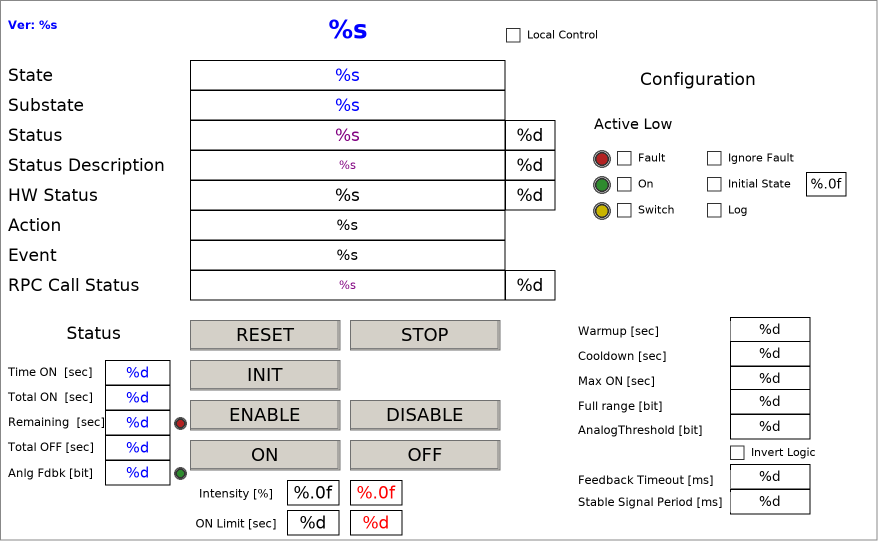
VISUALIZATION GUI_TEMPLATE_LAMP  // 878x541
VAR_IN_OUT
	m_Instance:	FB_LAMP;
END_VAR
    Rectangle (190,60 315x30), "%s", text variable: m_Instance.stat.sState
    Rectangle (190,90 315x30), "%s", text variable: m_Instance.stat.sSubstate
    Button (190,320 150x30), "RESET", input disabled if: (m_Instance.stat.bLocal = FALSE) <> 0
        OnMouseDown: execute { m_Instance.ctrl.nCommand := E_LAMP_COMMAND.RESET; m_Instance.ctrl.bExecute := TRUE; }
    Button (190,360 150x30), "INIT", input disabled if: (m_Instance.stat.bLocal = FALSE) <> 0
        OnMouseDown: execute { m_Instance.ctrl.nCommand := E_LAMP_COMMAND.INIT; m_Instance.ctrl.bExecute := TRUE; }
    Button (350,320 150x30), "STOP", input disabled if: (m_Instance.stat.bLocal = FALSE) <> 0
        OnMouseDown: execute { m_Instance.ctrl.nCommand := E_LAMP_COMMAND.STOP; m_Instance.ctrl.bExecute := TRUE; }
    Button (190,400 150x30), "ENABLE", input disabled if: (m_Instance.stat.bLocal = FALSE) <> 0
        OnMouseDown: execute { m_Instance.ctrl.nCommand := E_LAMP_COMMAND.ENABLE; m_Instance.ctrl.bExecute := TRUE; }
    Button (350,400 150x30), "DISABLE", input disabled if: (m_Instance.stat.bLocal = FALSE) <> 0
        OnMouseDown: execute { m_Instance.ctrl.nCommand := E_LAMP_COMMAND.DISABLE; m_Instance.ctrl.bExecute := TRUE; }
    Button (190,440 150x30), "ON", input disabled if: (m_Instance.stat.bLocal = FALSE) <> 0
        OnMouseDown: execute { m_Instance.ctrl.nCommand := E_LAMP_COMMAND.ON; m_Instance.ctrl.bExecute := TRUE; }
    Button (350,440 150x30), "OFF", input disabled if: (m_Instance.stat.bLocal = FALSE) <> 0
        OnMouseDown: execute { m_Instance.ctrl.nCommand := E_LAMP_COMMAND.OFF; m_Instance.ctrl.bExecute := TRUE; }
    Rectangle (5,60 180x30), "State"
    Rectangle (5,90 180x30), "Substate"
    Rectangle (190,120 315x30), "%s", text variable: m_Instance.stat.sStatus
    Rectangle (190,150 315x30), "%s", text variable: m_Instance.stat.sErrorText
    Rectangle (5,120 180x30), "Status"
    Rectangle (5,150 180x30), "Status Description"
    Rectangle (190,210 315x30), "%s", text variable: m_Instance.stat.sActionDesc
    Rectangle (190,240 315x30), "%s", text variable: m_Instance.stat.sEventDesc
    Rectangle (190,180 315x30), "%s", text variable: m_Instance.stat.sHwStatus
    Rectangle (5,180 180x30), "HW Status"
    Rectangle (505,180 50x30), "%d", text variable: m_Instance.stat.nHwStatus
    Rectangle (5,210 180x30), "Action"
    Rectangle (5,240 180x30), "Event"
    Rectangle (232,12 232x35), "%s", text variable: m_Instance.cfg.sName
    Rectangle (637,64 180x30), "Configuration"
    Rectangle (591,109 126x30), "Active Low"
    Checkbox (615,143 72x30), "Fault", variable: m_Instance.cfg.bActiveLowFault, input disabled if: (m_Instance.stat.bLocal = FALSE) <> 0
    Checkbox (705,143 102x30), "Ignore Fault", variable: m_Instance.cfg.bIgnoreFault, input disabled if: (m_Instance.stat.bLocal = FALSE) <> 0
    Checkbox (615,169 72x30), "On", variable: m_Instance.cfg.bActiveLowOn, input disabled if: (m_Instance.stat.bLocal = FALSE) <> 0
    Checkbox (615,195 72x30), "Switch", variable: m_Instance.cfg.bActiveLowSwitch, input disabled if: (m_Instance.stat.bLocal = FALSE) <> 0
    Checkbox (728,440 150x25), "Invert Logic", tooltip "If the logic is inverted, the lamp is considered to be ON, if the reading is below the threshold.", variable: m_Instance.cfg.bInvertAnalog, input disabled if: (m_Instance.stat.bLocal = FALSE) <> 0
    Rectangle (730,317 80x25), "%d", tooltip "Warmup time [sec] (>=0). Zero means no warmup.", text variable: m_Instance.cfg.nWarmup, input disabled if: (m_Instance.stat.bLocal = FALSE) <> 0
        OnMouseDown: write the text variable via Default, min 0
    Rectangle (575,321 155x20), "Warmup [sec]"
    Rectangle (575,346 155x20), "Cooldown [sec]"
    Rectangle (575,371 155x20), "Max ON [sec]"
    Rectangle (575,396 155x20), "Full range [bit]"
    Rectangle (730,341 80x25), "%d", tooltip "Cooldown time [sec] (>=0). Zero means no cooldown.", text variable: m_Instance.cfg.nCooldown, input disabled if: (m_Instance.stat.bLocal = FALSE) <> 0
        OnMouseDown: write the text variable via Default, min 0
    Rectangle (730,366 80x25), "%d", tooltip "Absolut maximum allowed time for lamp to be ON after last ON command [sec] (>=0). Zero means no limit. This is a safety feature.", text variable: m_Instance.cfg.nMaxOn, input disabled if: (m_Instance.stat.bLocal = FALSE) <> 0
        OnMouseDown: write the text variable via Default, min 0
    Rectangle (730,389 80x25), "%d", tooltip "Full range of A/D converter controlling the intensity [bit]. Examples: 12 bit A/D = 4095 15 bit A/D = 32767 16 bit A/D = 65535", text variable: m_Instance.cfg.nFullRange, input disabled if: (m_Instance.stat.bLocal = FALSE) <> 0
        OnMouseDown: write the text variable via Default, min 0
    Rectangle (730,414 80x25), "%d", tooltip "Analog feedback signal threshold [bit]. If used, the threshold should be > 0.", text variable: m_Instance.cfg.nAnalogThreshold, input disabled if: (m_Instance.stat.bLocal = FALSE) <> 0
        OnMouseDown: write the text variable via Default, min 0
    Rectangle (575,420 150x20), "AnalogThreshold [bit]"
    Rectangle (730,464 80x25), "%d", tooltip "When switching lamp ON, feedback signal should become active within this period.", text variable: m_Instance.cfg.nTimeout, input disabled if: (m_Instance.stat.bLocal = FALSE) <> 0
        OnMouseDown: write the text variable via Default, min 0
    Rectangle (575,470 155x20), "Feedback Timeout [ms]"
    Rectangle (287,480 52x25), "%.0f", tooltip "Set Lamp intensity [%] (0..100)", text variable: m_Instance.ctrl.lrIntensity, input disabled if: (m_Instance.stat.bLocal = FALSE) <> 0
        OnMouseDown: write the text variable via Default, min 0
    Rectangle (191,476 90x35), "Intensity [%]"
    Rectangle (350,480 52x25), "%.0f", tooltip "Actual Lamp intensity [%] (0..100)", text variable: m_Instance.stat.lrIntensity
    Checkbox (504,20 116x30), "Local Control", variable: m_Instance.stat.bLocal
    Rectangle (730,489 80x25), "%d", tooltip "A period of time [ms] that the feedback signal has to have constant value before taking its status. Minimum 10 ms.", text variable: m_Instance.cfg.nSigStablePeriod, input disabled if: (m_Instance.stat.bLocal = FALSE) <> 0
        OnMouseDown: write the text variable via Default, min 10
    Rectangle (575,492 155x20), "Stable Signal Period [ms]"
    Rectangle (48,318 92x30), "Status"
    Rectangle (105,360 65x25), "%d", tooltip "Time since last ON command [sec].", text variable: m_Instance.stat.nTimeOn
    Rectangle (105,385 65x25), "%d", tooltip "Total continuous time that Lamp has been ON [sec].", text variable: m_Instance.stat.nTimeOnTotal
    Rectangle (105,435 65x25), "%d", tooltip "Time since Lamp was switched OFF [sec].", text variable: m_Instance.stat.nTimeOff
    Rectangle (5,357 95x30), "Time ON [sec]"
    Rectangle (5,382 95x30), "Total ON [sec]"
    Rectangle (5,432 95x30), "Total OFF [sec]"
    Rectangle (505,120 50x30), "%d", tooltip "Device Status 0 - OK 1 - FAILURE", text variable: m_Instance.stat.nStatus
    Rectangle (190,270 315x30), "%s", text variable: m_Instance.stat.sRpcErrorText
    Rectangle (5,270 180x30), "RPC Call Status"
    Rectangle (5,10 99x30), "Ver: %s", tooltip "'IODev.library version'", text variable: m_Instance.stat.sLibVersion, input disabled if: true
    Rectangle (505,270 50x30), "%d", tooltip "RPC Error Code 0 - OK", text variable: m_Instance.stat.nRpcErrorCode
    Rectangle (505,150 50x30), "%d", tooltip "Error Code 0 - OK", text variable: m_Instance.stat.nErrorCode
    Lamp1 (592,149 20x20), tooltip "If ON, Fault signal is high (TRUE).", variable: m_Instance.i_bFault, style: Lamp-Lamp1-Red
    Lamp1 (592,201 20x20), tooltip "If ON, digital control output isignal s high (TRUE)", variable: m_Instance.q_bSwitch, style: Lamp-Lamp1-Yellow
    Lamp1 (592,175 20x20), tooltip "If ON, Lamp Digital feedback signal is high (TRUE).", variable: m_Instance.i_bOn, style: Lamp-Lamp1-Green
    Rectangle (287,510 52x25), "%d", tooltip "Set value for limit for Lamp to stay ON [sec] and automatically switch OFF. Zero means no limit.", text variable: m_Instance.ctrl.nTimeOnLimit, input disabled if: (m_Instance.stat.bLocal = FALSE) <> 0
        OnMouseDown: write the text variable via Default, min 0
    Rectangle (191,506 90x35), "ON Limit [sec]"
    Rectangle (350,510 52x25), "%d", tooltip "Actual Time ON limit [sec]", text variable: m_Instance.stat.nTimeOnLimit
    Rectangle (5,407 97x30), "Remaining [sec]"
    Rectangle (105,410 65x25), "%d", tooltip "Remaining time before the Lamp is switched OFF [sec].", text variable: m_Instance.stat.nTimeLeft
    Lamp1 (173,416 15x15), tooltip "If ON, check for maximum time is active.", variable: m_Instance.stat.bCheckTimeLeft, style: Lamp-Lamp1-Red
    Checkbox (705,169 100x30), "Initial State", tooltip "If selected, the lamp will switch ON on INIT.", variable: m_Instance.cfg.bInitialState, input disabled if: (m_Instance.stat.bLocal = FALSE) <> 0
    Rectangle (806,172 40x24), "%.0f", tooltip "Initial Intensity [%]", text variable: m_Instance.cfg.lrInitialIntensity, input disabled if: (m_Instance.stat.bLocal = FALSE) <> 0
        OnMouseDown: write the text variable via Default, min 0
    Checkbox (705,195 95x30), "Log", tooltip "Switch logging ON/OFF", variable: m_Instance.cfg.bLog, input disabled if: (m_Instance.stat.bLocal = FALSE) <> 0
    Lamp1 (173,466 15x15), tooltip "If ON, Lamp Analog feedback signal is active.", variable: m_Instance.stat.bOnAnalog, style: Lamp-Lamp1-Green
    Rectangle (105,460 65x25), "%d", tooltip "Analog Feedback [bit]", text variable: m_Instance.stat.nOn
    Rectangle (5,458 95x30), "Anlg Fdbk [bit]", tooltip "Analog Feedback [bit]"
END_VISUALIZATION

(* stored: Version 1.1.0.1, ProductVersion 3.1.4024.12
   Visu GUI_TEMPLATE_LAMP: Id {208abcb1-f1a3-4a00-92a5-f362cd7556ac} *)
